FUNCTION_BLOCK "GCS7_E_Maintanance1"	// FB 30
TITLE = Maintenance_1
//  
//COPYRIGHT:    (C) 1997  BUHLER AG, CH-9240 UZWIL, SWITZERLAND
//
//PRODUCT:      GCS7
//
//TITLE:        Element Control Maintenance 1
//
//-------------------------------------------------------------------------
//
//IDENT:        AUTHOR:             DEPT:                       DATE:
//
//FB30.2.2      Ph. Engler          GP92                        31-Jul-2009
//              Flags GCS7_Gr_InMaintWarning and GCS7_Gr_InMaintFault
//FB30.2.1      A. Egli             CT3                         18-Aug-2003
//              FDefineValue 
//FB30.2.0      A. Egli             CT3                         17-Jun-2002
//              New Release with one block 
//FB30.1.1      A.Egli              CT3                         04-Mar-2002
//              Reset CmdFaultReset
//FB30.1.0      A.Egli              CT3                         20-Mar-2000
//              1st Release in S7
//
//-------------------------------------------------------------------------
//
//PURPOSE:      MANUAL : see [MAIN1xxMAN]
//
//RESTRICTIONS: S7
//              ACCU2: Pointer to dynamic datas of the element
//              ACCU1: Pointer to parameter datas of the element
//
//-------------------------------------------------------------------------
//=======================================================
//Log Message: 
//------------------------------------------------------
//1   Counter cleared
//9   fault cancelled
//11  fault 
//12  warning 
//
//=======================================================
//StCode:  State               
//------------------------------------------------------
// 32   StFault        
//  2   StWarning      
//  3   StNormal       
//
//
AUTHOR : EA
FAMILY : GCS7LL
NAME : Maintena
VERSION : 2.2
VAR
  StCode : INT ;	//Element state code
  spare0200 : BOOL ;
  spare0201 : BOOL ;
  spare0202 : BOOL ;
  spare0203 : BOOL ;
  spare0204 : BOOL ;
  InpFault : BOOL ;	//Input to count OutFaultCnt
  InpCount : BOOL ;	//Input to count OutValue
  spare0207 : BOOL ;
  CmdClearValue : BOOL ;	//Clear values
  spare0301 : BOOL ;
  spare0302 : BOOL ;
  CmdFaultReset : BOOL ;	//Command fault reset
  spare0304 : BOOL ;
  spare0305 : BOOL ;
  spare0306 : BOOL ;
  spare0307 : BOOL ;
  OutCopyCount : BOOL ;	//Copy of InpCount
  OutCopyFault : BOOL ;	//Copy of InpFault
  spare0402 : BOOL ;
  spare0403 : BOOL ;
  spare0404 : BOOL ;
  spare0405 : BOOL ;
  spare0406 : BOOL ;
  spare0407 : BOOL ;
  spare0500 : BOOL ;
  spare0501 : BOOL ;
  StNormal : BOOL ;	//OutValue < InWarningValue
  StWarning : BOOL ;	//OutValue >=InWarningValue
  StFault : BOOL ;	//OutValue >=InFaultValue
  spare0505 : BOOL ;
  spare0506 : BOOL ;
  spare0507 : BOOL ;
  InFaultLimit : DINT ;	//Limit for fault           [0.1h] or [number]
  InWarningLimit : DINT ;	//Limit for warning         [0.1h] or [number]
  OutValue : DINT ;	//Actual maintenance value  [0.1h] or [number]
  OutFaultCnt : INT ;	//Number of fault of monitored object [number]
  OutCountSec : INT ;	//Help value to count second
  OutAlarmNrLog : INT ;	//Last textnumber send to log
  Par : STRUCT
   ParObjectNo : INT ;	//Is used for communication with PC, e.g. for message
   ParMsgType : INT ;	//Is used for message (translation of state)
   ParHornCode : INT ;	//Is used by horn module
   ParLogOff : BOOL ;	//Report is off
   ParSpare0401 : BOOL ;
   ParEdgeCnt : BOOL ;	//Type is flag counter
  END_STRUCT ;
END_VAR
VAR_TEMP
  tmpLOGvalue : WORD ;	//LOG value
  tmpLenDyn : DINT ;
  tmpReport : BOOL ;	//Global LOG all
  tmpLocal : BOOL ;
  tmpWarning : BOOL ;
  tmpFault : BOOL ;
END_VAR
BEGIN
NETWORK
TITLE =  Start Global
      L     30;
      T     #tmpLenDyn;	//--> Len dynamic data in byte
NETWORK
TITLE = PC Control
//=== Test Object number =====================
      L     "SYS_DirectCtrlDB".PC.ObjectNo;	//PCControl.ObjectNo
      L     #Par.ParObjectNo;	//Input ObjectNo
      <>I;
      JC    Ctrl;
//=== Test OType      ========================
      L     1830;	//Input object type
      L     "SYS_DirectCtrlDB".PC.ObjectType;	//PCControl.ObjectType
      <>I;
      JC    Ctrl;
//=== Test Handshake =========================
      A     "SYS_DirectCtrlDB".PC.Hsk.FExamine;	// Handshake.FExamine
      JC    pExa;
      A     "SYS_DirectCtrlDB".PC.Hsk.FDefineCmd;	// Handshake.FDefineCmd
      O     "SYS_DirectCtrlDB".PC.Hsk.FDefineValue;	// PC.Hsk.FDefineValue     //[2.1]
      JC    pCmd;
      A     "SYS_DirectCtrlDB".PC.Hsk.FDefinePara;	// Handshake.FDefinePara
      JC    pPar;
pIni: L     2;	// FcInit
      UC    "SYS_DirectCtrl";
      JU    Ctrl;
// Write parameter
pPar: NOP   0;
// Write new commands from PC to Interface of group 
pCmd: A     "SYS_DirectCtrlDB".PC.Cmd1[8];	//Cmd1[8] =CmdClearValue
      S     #CmdClearValue;
      A     "SYS_DirectCtrlDB".PC.Cmd1[11];	//Cmd1[11] =CmdFaultReset
      S     #CmdFaultReset;
//Define Value
      AN    "SYS_DirectCtrlDB".PC.Hsk.FDefineValue;	// PC.Hsk.FDefineValue
      JC    pIni;
      LAR1  P#DBX 58.0;	//PCControl.Value[1]
      L     DBD [AR1,P#6.0];	//PCControl.Value[x+3]
      T     #InFaultLimit;
      L     DBD [AR1,P#10.0];	//PCControl.Value[x+5]
      T     #InWarningLimit;
      JU    pIni;
pExa: TAR2;	// Address Dynamic datas
      T     "SYS_DirectCtrlDB".GC.InDynAddr;	// -->PCControl.GC.InDynAddr
      L     #tmpLenDyn;	// Length Dynamic datas
      T     "SYS_DirectCtrlDB".GC.InDynLen;	// -->PCControl.GC.InDynLen
      L     0;
      T     "SYS_DirectCtrlDB".GC.InParaAddr;	// -->PCControl.GC.InParaAddr
      T     "SYS_DirectCtrlDB".GC.InParaLen;	// -->PCControl.GC.InParaLen
      L     1;	// Code FcExamine
      UC    "SYS_DirectCtrl";
      L     10;	//Revision
      T     "SYS_DirectCtrlDB".GC.Revision;
Ctrl: NOP   0;
NETWORK
TITLE =  All State Init
//---FaultReset is on---
      A     "GCS7_Gr_OutFaultReset";	//Gr.OutFaultReset
      S     #CmdFaultReset;
//===Clear tmp Variable
      AN    #CmdClearValue;
      JC    glJ1;
      L     0;
      T     #OutValue;
      T     #OutFaultCnt;
      T     #OutCountSec;
      O     #Par.ParLogOff;	//---Set LOG Message
      JC    glJ1;
      L     B#(3, 7);	// Message ('Value Cleared' )
      T     #tmpLOGvalue;
      L     W#16#FF;
      AW;
      T     #OutAlarmNrLog;
      CALL  "GCS7_LogConvert" (
           ObjectNo                 := #Par.ParObjectNo,
           MsgType                  := #Par.ParMsgType,
           ClassMsgTxt              := #tmpLOGvalue,
           OType                    := 1030);	// LOG Message Converter / Entry / Contains Class and TextNo
//===Global Group Orders===
//==Count Edges
glJ1: AN    #Par.ParEdgeCnt;
      JC    glJ2;
      A     #InpCount;
      FP    #OutCopyCount;
      JC    glIc;
      JU    glJ4;
//==Running time
glJ2: AN    "GCS7_Gr_OutTick1s";	//Gr.OutTick1s
      ON    #InpCount;
      JC    glJ4;
      L     #OutCountSec;
      +     1;
      T     #OutCountSec;
      L     360;
      <I;
      JC    glJ4;
glIc: L     #OutValue;
      +     L#1;
      T     #OutValue;
      L     0;
      T     #OutCountSec;
//==Count faults
glJ4: NOP   0;
      A     #InpFault;
      FP    #OutCopyFault;
      JCN   glJ5;
      L     #OutFaultCnt;
      +     1;
      T     #OutFaultCnt;
//===Help flags
glJ5: NOP   0;
      L     #OutValue;
      L     #InWarningLimit;
      >=D;
      A(;
      L     0;
      <>D;
      );
      =     #tmpWarning;
      L     #OutValue;
      L     #InFaultLimit;
      >=D;
      A(;
      L     0;
      <>D;
      );
      =     #tmpFault;
NETWORK
TITLE = States
//===State machine===
      A     #StNormal;
      JC    S2;
      A     #StWarning;
      JC    S3;
      A     #StFault;
      JC    S4;
      S     #StNormal;	// Init
      JU    S2;
NETWORK
TITLE = StNormal
// Any transition to StNormal
      S     #StNormal;
      JU    LOG;
//=== Logic ====
//Transition to StFault
S2:   A     #tmpFault;
      R     #StNormal;
      JC    xxS4;
//Transition to StWarning
      A     #tmpWarning;
      R     #StNormal;
      JC    xxS3;
      JU    OUT;
NETWORK
TITLE = StWarning
// Any transition to StWarning
xxS3: S     #StWarning;
      L     B#(1, 12);	// Message ('Warning')
      JU    LOG;
//=== Logic ====
// Transition to StFault
S3:   A     #tmpFault;
      R     #StWarning;
      JC    xxS4;
//  Retry message
      A     #CmdFaultReset;
      O     "GCS7_Gr_OutFaultReset";	// OutFaultReset
      A     #tmpWarning;
      JC    xxS3;
// Transition to StNormal
      A     #tmpWarning;
      JC    OUT;
      R     #StWarning;
      S     #StNormal;
      L     B#(3, 9);	// Message ('fault cancelled' )
      JU    LOG;
NETWORK
TITLE = StFault
// Any transiton to Fault  
xxS4: S     "GCS7_Gr_InFaultFlag";	// Gr.InFaultFlag
      S     #StFault;
      CALL  "SYS_Horn_Code" (
           FcCode                   := 1,
           ParObjectType            := 1030,
           ParObjectNo              := #Par.ParObjectNo,
           ParHornCode              := #Par.ParHornCode);
      L     B#(1, 11);	// Message ('fault')
      JU    LOG;
//=== Logic ====
// retry of fault message
S4:   A     #CmdFaultReset;
      O     "GCS7_Gr_OutFaultReset";	//Gr.OutFaultReset
      A     #tmpFault;
      L     B#(1, 11);	// Message ('fault')
      JC    LOG;
      A     #tmpFault;
      JC    OUT;
      R     #StFault;
      S     #StNormal;
      L     B#(3, 9);	// Message ('fault cancelled' )
      JU    LOG;
NETWORK
TITLE = LOG
LOG:  A     #Par.ParLogOff;	//---Set LOG Message
      JC    OUT;
      T     #tmpLOGvalue;
      L     W#16#FF;
      AW;
      T     #OutAlarmNrLog;
      CALL  "GCS7_LogConvert" (
           ObjectNo                 := #Par.ParObjectNo,
           MsgType                  := #Par.ParMsgType,
           ClassMsgTxt              := #tmpLOGvalue,
           OType                    := 1030);	// LOG Message Converter / Entry / Contains Class and TextNo
NETWORK
TITLE = Global End
OUT:  SET;
      R     #CmdClearValue;
      R     #CmdFaultReset;	//[1.1]
// 
      A     #StWarning;	//[2.2]
      S     "GCS7_Gr_InMaintWarning";	//[2.2]
      A     #StFault;	//[2.2]
      S     "GCS7_Gr_InMaintFault";	//[2.2]
NETWORK
TITLE = State Code
      L     2;	// Code: Warning
      A     #StWarning;
      JC    STC;
      L     3;	// Code: Normal
      A     #StNormal;
      JC    STC;
      L     32;	// Code: fault
STC:  L     #StCode;	// Old state code
      TAK;
      T     #StCode;	// Save state code
      <>I;
      L     3;	// Load code for CBit methode
      CC    "SYS_CBitCtrl";
END_FUNCTION_BLOCK

FUNCTION_BLOCK "GCS7_E_Maintanance2"	// FB 31
TITLE = Maintenance_2
//  
//COPYRIGHT:    (C) 1997  BUHLER AG, CH-9240 UZWIL, SWITZERLAND
//
//PRODUCT:      GCS7
//
//TITLE:        Element Control Maintenance 2
//
//-------------------------------------------------------------------------
//
//IDENT:        AUTHOR:             DEPT:                       DATE:
//
//FB31.2.2      Ph. Engler          GP92                        31-Jul-2009
//              Flags GCS7_Gr_InMaintWarning and GCS7_Gr_InMaintFault
//FB31.2.1      A. Egli             CT3                         18-Aug-2003
//              FDefineValue
//FB31.2.0      A. Egli             CT3                         17-Jun-2002
//              New Release with one block 
//FB31.1.1      A.Egli              CT3                         04-Mar-2002
//              Reset CmdFaultReset
//FB31.1.0      A.Egli              CT3                         20-Mar-2000
//              1st Release in S7
//
//-------------------------------------------------------------------------
//
//PURPOSE:      MANUAL : see [MAIN2xxMAN]
//                
//
//RESTRICTIONS: S7
//              ACCU2: Pointer to dynamic datas of the element
//              ACCU1: Pointer to parameter datas of the element
//
//-------------------------------------------------------------------------
//=======================================================
//Log Message: 
//------------------------------------------------------
// 1   Counter cleared
// 9   fault cancelled
//11   fault 
//12   warning 
//
//
//=======================================================
//StCode:  State               
//------------------------------------------------------
// 32   StFault        
//  2   StWarning      
//  3   StNormal       
//
AUTHOR : EA
FAMILY : GCS7LL
NAME : Maintena
VERSION : 2.2
VAR
  StCode : INT ;	//Element state code
  spare0200 : BOOL ;
  spare0201 : BOOL ;
  spare0202 : BOOL ;
  spare0203 : BOOL ;
  spare0204 : BOOL ;
  InpFault : BOOL ;	//Input to count fault values
  InpRun : BOOL ;	//Input to count running times
  spare0207 : BOOL ;
  CmdClearValue : BOOL ;	//Clear maintenance values
  CmdClearTotalValue : BOOL ;	//Clear maintenance values and total hours
  spare0302 : BOOL ;
  CmdFaultReset : BOOL ;	//Command fault reset
  spare0304 : BOOL ;
  spare0305 : BOOL ;
  spare0306 : BOOL ;
  spare0307 : BOOL ;
  OutCopyFault : BOOL ;	//Copy of InpFault
  spare0401 : BOOL ;
  spare0402 : BOOL ;
  spare0403 : BOOL ;
  spare0404 : BOOL ;
  spare0405 : BOOL ;
  spare0406 : BOOL ;
  spare0407 : BOOL ;
  spare0500 : BOOL ;
  spare0501 : BOOL ;
  StNormal : BOOL ;	//OutValue < InWarningValue
  StWarning : BOOL ;	//OutValue >=InWarningValue
  StFault : BOOL ;	//OutValue >=InFaultValue
  spare0505 : BOOL ;
  spare0506 : BOOL ;
  spare0507 : BOOL ;
  InFaultLimit : DINT ;	//Limit for fault      [0.1 h]
  InWarningLimit : DINT ;	//Limit for warning    [0.1 h]
  OutTotalHours : DINT ;	//Running hours since last maintenance [0.1 h]
  OutMaintenanceHours : DINT ;	//Running hours since last maintenance [0.1 h]
  OutFaultHours : DINT ;	//Fault hours since last maintenance [0.1 h]
  OutFaultCounter : INT ;
  OutResetDate : STRUCT 	//Last maintenance
   Year : INT ;
   Month : BYTE ;
   Day : BYTE ;
   Hour : BYTE ;
   Min : BYTE ;
  END_STRUCT ;
  OutTotalSec : INT ;	//Help value to count seconds
  OutMaintenanceSec : INT ;	//Help value to count seconds
  OutFaultSec : INT ;	//Help value to count seconds
  OutAlarmNrLog : INT ;	//Last textnumber send to log
  Par : STRUCT
   ParObjectNo : INT ;	//Is used for communication with PC, e.g. for message
   ParMsgType : INT ;	//Is used for message (translation of state)
   ParHornCode : INT ;	//Is used by horn module
   ParLogOff : BOOL ;	//Report is off
  END_STRUCT ;
END_VAR
VAR_TEMP
  tmpLOGvalue : WORD ;	//LOG value
  tmpLenDyn : DINT ;
  tmpReport : BOOL ;	//Global LOG all
  tmpLocal : BOOL ;
  tmpWarning : BOOL ;
  tmpFault : BOOL ;
  tmpDateTime : DATE_AND_TIME ;
  tmpRet : INT ;
END_VAR
BEGIN
NETWORK
TITLE =  Start Global
      L     48;
      T     #tmpLenDyn;	//--> Len dynamic data in byte
NETWORK
TITLE = PC Control
//=== Test Object number =====================
      L     "SYS_DirectCtrlDB".PC.ObjectNo;	//PCControl.ObjectNo
      L     #Par.ParObjectNo;	//Input ObjectNo
      <>I;
      JC    Ctrl;
//=== Test OType      ========================
      L     1831;	//Input object type
      L     "SYS_DirectCtrlDB".PC.ObjectType;	//PCControl.ObjectType
      <>I;
      JC    Ctrl;
//=== Test Handshake =========================
      A     "SYS_DirectCtrlDB".PC.Hsk.FExamine;	// Handshake.FExamine
      JC    pExa;
      A     "SYS_DirectCtrlDB".PC.Hsk.FDefineCmd;	// Handshake.FDefineCmd
      O     "SYS_DirectCtrlDB".PC.Hsk.FDefineValue;	// Handshake.FDefineValue  //[2.1]
      JC    pCmd;
      A     "SYS_DirectCtrlDB".PC.Hsk.FDefinePara;	// Handshake.FDefinePara
      JC    pPar;
pIni: L     2;	// FcInit
      UC    "SYS_DirectCtrl";
      JU    Ctrl;
// Write parameter
pPar: NOP   0;
// Write new commands from PC to Interface of group 
pCmd: A     "SYS_DirectCtrlDB".PC.Cmd1[8];	//Cmd1[8] =CmdClearValue
      S     #CmdClearValue;
      A     "SYS_DirectCtrlDB".PC.Cmd1[9];	//Cmd1[8] =CmdClearValue
      S     #CmdClearTotalValue;
      A     "SYS_DirectCtrlDB".PC.Cmd1[11];	//Cmd1[11] =CmdFaultReset
      S     #CmdFaultReset;
//Define Value
      AN    "SYS_DirectCtrlDB".PC.Hsk.FDefineValue;	// PC.Hsk.FDefineValue
      JC    pIni;
      LAR1  P#DBX 58.0;	//PCControl.Value[1]
      L     DBD [AR1,P#6.0];	//PCControl.Value[x+3]
      T     #InFaultLimit;
      L     DBD [AR1,P#10.0];	//PCControl.Value[x+5]
      T     #InWarningLimit;
      JU    pIni;
pExa: TAR2;	// Address Dynamic datas
      T     "SYS_DirectCtrlDB".GC.InDynAddr;	// -->PCControl.GC.InDynAddr
      L     #tmpLenDyn;	// Length Dynamic datas
      T     "SYS_DirectCtrlDB".GC.InDynLen;	// -->PCControl.GC.InDynLen
      L     0;
      T     "SYS_DirectCtrlDB".GC.InParaAddr;	// -->PCControl.GC.InParaAddr
      T     "SYS_DirectCtrlDB".GC.InParaLen;	// -->PCControl.GC.InParaLen
      L     1;	// Code FcExamine
      UC    "SYS_DirectCtrl";
      L     10;	//Revision
      T     "SYS_DirectCtrlDB".GC.Revision;
Ctrl: NOP   0;
NETWORK
TITLE =  All State Init
//---FaultReset is on--
      A     "GCS7_Gr_OutFaultReset";	//Gr.OutFaultReset
      S     #CmdFaultReset;
//===Clear tmp Variable
      AN    #CmdClearTotalValue;
      JC    glR0;
      L     0;
      T     #OutTotalHours;
      T     #OutTotalSec;
      O     #Par.ParLogOff;	//---Set LOG Message
      JC    glR0;
      L     B#(3, 8);	// Message ('Total Value Cleared' )
      T     #tmpLOGvalue;
      L     W#16#FF;
      AW;
      T     #OutAlarmNrLog;
      CALL  "GCS7_LogConvert" (
           ObjectNo                 := #Par.ParObjectNo,
           MsgType                  := #Par.ParMsgType,
           ClassMsgTxt              := #tmpLOGvalue,
           OType                    := 1031);	// LOG Message Converter / Entry / Contains Class and TextNo
//===Clear tmp Variable
glR0: AN    #CmdClearValue;
      JC    glJ1;
      CALL  "SIEMENS_READ_CLK" (
           RET_VAL                  := #tmpRet,
           CDT                      := #tmpDateTime);
      LAR1  P##tmpDateTime;
      L     1900;
      L     LB [AR1,P#0.0];
      BTI;
      +I;
      L     1990;
      >=I;
      TAK;
      JC    glJa;
      +     100;
glJa: T     #OutResetDate.Year;
      L     LB [AR1,P#1.0];
      BTI;
      T     #OutResetDate.Month;
      L     LB [AR1,P#2.0];
      BTI;
      T     #OutResetDate.Day;
      L     LB [AR1,P#3.0];
      BTI;
      T     #OutResetDate.Hour;
      L     LB [AR1,P#4.0];
      BTI;
      T     #OutResetDate.Min;
      L     #OutMaintenanceHours;
      L     0;
      ==D;
      T     #OutMaintenanceHours;
      T     #OutFaultHours;
      T     #OutFaultCounter;
      T     #OutMaintenanceSec;
      T     #OutFaultSec;
      O     #Par.ParLogOff;	//---Set LOG Message
      JC    glJ1;
      L     B#(3, 7);	// Message ('Value Cleared' )
      T     #tmpLOGvalue;
      L     W#16#FF;
      AW;
      T     #OutAlarmNrLog;
      CALL  "GCS7_LogConvert" (
           ObjectNo                 := #Par.ParObjectNo,
           MsgType                  := #Par.ParMsgType,
           ClassMsgTxt              := #tmpLOGvalue,
           OType                    := 1031);	// LOG Message Converter / Entry / Contains Class and TextNo
//===Global Group Orders===
// Count Faults
glJ1: A     #InpFault;
      FP    #OutCopyFault;
      JCN   glJ2;
      L     #OutFaultCounter;
      +     L#1;
      T     #OutFaultCounter;
// Count Fault time
glJ2: AN    "GCS7_Gr_OutTick1s";	//Gr.OutTick1s
      ON    #InpFault;
      JC    glJ3;
      L     #OutFaultSec;
      +     1;
      T     #OutFaultSec;
      L     360;
      <I;
      JC    glJ3;
      L     #OutFaultHours;
      +     L#1;
      T     #OutFaultHours;
      L     0;
      T     #OutFaultSec;
//Maintenance hour
glJ3: AN    "GCS7_Gr_OutTick1s";	//Gr.OutTick1s
      ON    #InpRun;
      JC    glJ4;
      L     #OutMaintenanceSec;
      +     1;
      T     #OutMaintenanceSec;
      L     360;
      <I;
      JC    glJ4;
      L     #OutMaintenanceHours;
      +     L#1;
      T     #OutMaintenanceHours;
      L     0;
      T     #OutMaintenanceSec;
//Total hour
glJ4: AN    "GCS7_Gr_OutTick1s";	//Gr.OutTick1s
      ON    #InpRun;
      JC    glJ5;
      L     #OutTotalSec;
      +     1;
      T     #OutTotalSec;
      L     360;
      <I;
      JC    glJ5;
      L     #OutTotalHours;
      +     L#1;
      T     #OutTotalHours;
      L     0;
      T     #OutTotalSec;
//Help Flags
glJ5: L     #OutMaintenanceHours;
      L     #InWarningLimit;
      >=D;
      A(;
      L     0;
      <>D;
      );
      =     #tmpWarning;
      L     #OutMaintenanceHours;
      L     #InFaultLimit;
      >=D;
      A(;
      L     0;
      <>D;
      );
      =     #tmpFault;
NETWORK
TITLE = States
//===State machine===
      A     #StNormal;
      JC    S2;
      A     #StWarning;
      JC    S3;
      A     #StFault;
      JC    S4;
      S     #StNormal;	// Init
      JU    S2;
NETWORK
TITLE = StNormal
// Any transition to StNormal
      S     #StNormal;
      JU    LOG;
//=== Logic ====
//Transition to StFault
S2:   A     #tmpFault;
      R     #StNormal;
      JC    xxS4;
//Transition to StWarning
      A     #tmpWarning;
      R     #StNormal;
      JC    xxS3;
      JU    OUT;
NETWORK
TITLE = StWarning
// Any transition to StWarning
xxS3: S     #StWarning;
      L     B#(1, 12);	// Message ('Warning')
      JU    LOG;
//=== Logic ====
// Transition to StFault
S3:   A     #tmpFault;
      R     #StWarning;
      JC    xxS4;
//  Retry message
      A     #CmdFaultReset;
      O     "GCS7_Gr_OutFaultReset";	// OutFaultReset
      A     #tmpWarning;
      JC    xxS3;
// Transition to StNormal
      A     #tmpWarning;
      JC    OUT;
      R     #StWarning;
      S     #StNormal;
      L     B#(3, 9);	// Message ('fault cancelled' )
      JU    LOG;
NETWORK
TITLE = StFault
// Any transiton to Fault  
xxS4: S     "GCS7_Gr_InFaultFlag";	// Gr.InFaultFlag
      S     #StFault;
      CALL  "SYS_Horn_Code" (
           FcCode                   := 1,
           ParObjectType            := 1031,
           ParObjectNo              := #Par.ParObjectNo,
           ParHornCode              := #Par.ParHornCode);
      L     B#(1, 11);	// Message ('fault')
      JU    LOG;
//=== Logic ====
// retry of fault message
S4:   A     #CmdFaultReset;
      O     "GCS7_Gr_OutFaultReset";	//Gr.OutFaultReset
      A     #tmpFault;
      L     B#(1, 11);	// Message ('fault')
      JC    LOG;
      A     #tmpFault;
      JC    OUT;
      R     #StFault;
      S     #StNormal;
      L     B#(3, 9);	// Message ('fault cancelled' )
      JU    LOG;
NETWORK
TITLE = LOG
LOG:  A     #Par.ParLogOff;	//---Set LOG Message
      JC    OUT;
      T     #tmpLOGvalue;
      L     W#16#FF;
      AW;
      T     #OutAlarmNrLog;
      CALL  "GCS7_LogConvert" (
           ObjectNo                 := #Par.ParObjectNo,
           MsgType                  := #Par.ParMsgType,
           ClassMsgTxt              := #tmpLOGvalue,
           OType                    := 1031);	// LOG Message Converter / Entry / Contains Class and TextNo
NETWORK
TITLE = Global End
OUT:  SET;
      R     #CmdClearValue;
      R     #CmdClearTotalValue;
      R     #CmdFaultReset;	//[1.1]
// 
      A     #StWarning;	//[2.2]
      S     "GCS7_Gr_InMaintWarning";	//[2.2]
      A     #StFault;	//[2.2]
      S     "GCS7_Gr_InMaintFault";	//[2.2]
NETWORK
TITLE = State Code
      L     2;	// Code: Warning
      A     #StWarning;
      JC    STC;
      L     3;	// Code: Normal
      A     #StNormal;
      JC    STC;
      L     32;	// Code: fault
STC:  L     #StCode;	// Old state code
      TAK;
      T     #StCode;	// Save state code
      <>I;
      L     3;	// Load code for CBit methode
      CC    "SYS_CBitCtrl";
END_FUNCTION_BLOCK

FUNCTION_BLOCK "GCS7_E_MZAF"	// FB 32
TITLE = Flowbalancer MZAF
//  
//COPYRIGHT:    (C) 1997  BUHLER AG, CH-9240 UZWIL, SWITZERLAND
//
//PRODUCT:      GCS7
//
//TITLE:        Element Control MZAF
//
//-------------------------------------------------------------------------
//
//IDENT:        AUTHOR:             DEPT:                       DATE:
//
//FB32.3.0      A. Egli             CT3                         17-Jun-2002
//              New Release with one block 
//FB32.2.1      A. Egli             CT3                         11-Oct-1999
//              M12.2 "Gr.OutCmdNext removed
//FB32.2A       A. Egli             CT3                         04-Mai-1998
//              StFault = StCode 32
//FB32.1A       A.Egli              AEE61                       31-Jul-1997
//              1st Release in S7
//
//-------------------------------------------------------------------------
//
//PURPOSE:      MANUAL : see [MZAxxMAN]
//
//RESTRICTIONS: S7
//              ACCU2: Pointer to dynamic datas of the element
//              ACCU1: Pointer to parameter datas of the element
//
//-------------------------------------------------------------------------
//
//=======================================================
//Log Message: 
//------------------------------------------------------
// 0   stopped
// 1   started
// 9   fault cancelled
//10  fault adjust
//
//=======================================================
//StCode:  State               
//------------------------------------------------------
//32   StFault                 
// 1   StStopped                    Stopped
//41   Stopped.HWStop               StStopped + InHWStop 
//51   Stopped.DPFault              StStopped + DPFault
// 2   StAdjusting             
// 3   StStarted               
//
//
//
AUTHOR : EA
FAMILY : GCS7LL
NAME : MZAF
VERSION : 3.0
VAR
  StCode : INT ;	//Element state code
  InEnable : BOOL ;	//Enable to run
  spare0201 : BOOL ;
  spare0202 : BOOL ;
  spare0203 : BOOL ;
  spare0204 : BOOL ;
  CmdNewJob : BOOL ;	//Pulse to erase OutJobWeight
  InFlapOpen : BOOL ;	//Flap is open, command to count up OutJobWeight
  InpAdjusted : BOOL ;	//Digital input element is adjusted
  CmdOff : BOOL ;	//Pulse to start in manual mode
  CmdOn : BOOL ;	//Pulse to stop in manual mode
  CmdNext : BOOL ;	//Start next element (Automatic mode)
  CmdFaultReset : BOOL ;	//Command to reset fault
  InLocal : BOOL ;	//1= Local mode
  InManual : BOOL ;	//1= Manual/ 0= Automatic
  InReport : BOOL ;	//Report of all state transitions
  spare0307 : BOOL ;
  InHWStop : BOOL ;	//ALL : HW stop is detected, no fault
  InDPFault : BOOL ;	//ALL : DP-Fault is detected, no fault
  spare0402 : BOOL ;
  spare0403 : BOOL ;
  spare0404 : BOOL ;
  spare0405 : BOOL ;
  spare0406 : BOOL ;
  OutpAirValve : BOOL ;	//Digital output air valve
  StStopped : BOOL ;	//Element is stopped
  StAdjusting : BOOL ;	//Element is adjusting
  StStarted : BOOL ;	//Element is adjusted
  spare0503 : BOOL ;
  StFault : BOOL ;	//Element has a fault
  InOutFlowratePpm : INT ;	//Flowrate target value in [0.1 %]
  InOutFlowrate : DINT ;	//Flowrate target value in [kg/h]
  OutJobWeight : DINT ;	//Total feeded weight [kg]
  OutpFlowrate : INT ;	//Analog value to set flowrate [digits]
  OutAlarmNrLog : INT ;	//Last textnumber send to log
  Par : STRUCT
   ParObjectNo : INT ;	//Is used for communication with PC, e.g. for message
   ParMsgType : INT ;	//Is used for message (translation of state)
   ParHornCode : INT ;	//Is used by horn module
   ParLogOff : BOOL ;	//Report is off
   ParManual : BOOL ;	//Manual mode without interlocking
   ParFlowratePc : BOOL ;	//Target value for flowrate in Pc
   ParSpare0403 : BOOL ;
   ParWago : BOOL ;	//Wago analog module format
   ParMonTime : INT ;	//After this time the element must be adjusted [0.1 s]
   ParFlowrate100Pc : DINT  := L#10000;	//Flow rate by 100 % of analog output [kg/h]
   OutMonTime : INT  := 100;	//Actual monitoring time [0.1 s]
   OutWtCorrection : REAL ;	//Correction weight for calcuation of OutWtTotal [kg]
  END_STRUCT ;
END_VAR
VAR_TEMP
  tmpLOGvalue : WORD ;	//LOG value
  tmpLenDyn : DINT ;
  tmpReport : BOOL ;	//Global LOG all
  tmpEnable : BOOL ;
  tmpEndTime : BOOL ;
  tmpLocal : BOOL ;
  tmpMaxDigits : REAL ;	//ParWago=0: 27'648 / ParWago=1: 32'767
  tmpLocalFault : BOOL ;
END_VAR
BEGIN
NETWORK
TITLE =  Start Global
      L     38;
      T     #tmpLenDyn;	//--> Len dynamic data in byte
NETWORK
TITLE = PC Control
//=== Test Object number =====================
      L     "SYS_DirectCtrlDB".PC.ObjectNo;	//PCControl.ObjectNo
      L     #Par.ParObjectNo;	//Input ObjectNo
      <>I;
      JC    Ctrl;
//=== Test OType      ========================
      L     1032;	//Input object type
      L     "SYS_DirectCtrlDB".PC.ObjectType;	//PCControl.ObjectType
      <>I;
      JC    Ctrl;
//=== Test Handshake =========================
      A     "SYS_DirectCtrlDB".PC.Hsk.FExamine;	// Handshake.FExamine
      JC    pExa;
      A     "SYS_DirectCtrlDB".PC.Hsk.FDefineCmd;	// Handshake.FDefineCmd
      JC    pCmd;
      A     "SYS_DirectCtrlDB".PC.Hsk.FDefinePara;	// Handshake.FDefinePara
      JC    pPar;
pIni: L     2;	// FcInit
      UC    "SYS_DirectCtrl";
      JU    Ctrl;
// Write parameter 
pPar: LAR1  P#DBX 58.0;	//PCControl.Value[1]
      L     #tmpLenDyn;
      SLD   3;
      +AR1;
      L     DBW [AR1,P#8.0];	//PCControl.Value
      T     #Par.ParMonTime;
// Write new commands from PC to Interface of group 
pCmd: A     "SYS_DirectCtrlDB".PC.Cmd1[8];	//Cmd1[8] =CmdOff
      S     #CmdOff;
      A     "SYS_DirectCtrlDB".PC.Cmd1[9];	//Cmd1[9] =CmdOn
      S     #CmdOn;
      A     "SYS_DirectCtrlDB".PC.Cmd1[10];	//Cmd1[10] =CmdNext
      S     #CmdNext;
      A     "SYS_DirectCtrlDB".PC.Cmd1[11];	//Cmd1[11] =CmdFaultReset
      S     #CmdFaultReset;
      A     "SYS_DirectCtrlDB".PC.Cmd1[13];	//Cmd1[13] =CmdManualOn
      S     #InManual;
      A     "SYS_DirectCtrlDB".PC.Cmd2[13];	//Cmd2[13] =CmdManualOff
      R     #InManual;
      A     "SYS_DirectCtrlDB".PC.Cmd1[14];	//Cmd1[14]=CmdReportOn
      S     #InReport;
      A     "SYS_DirectCtrlDB".PC.Cmd2[14];	//Cmd2[14]=CmdReportOff
      R     #InReport;
//Define Value
      AN    "SYS_DirectCtrlDB".PC.Hsk.FDefineValue;	// PC.Hsk.FDefineValue
      ON    #InManual;
      JC    pIni;
      LAR1  P#DBX 58.0;
      L     DBW [AR1,P#6.0];
      T     #InOutFlowratePpm;
      L     DBD [AR1,P#8.0];
      T     #InOutFlowrate;
      JU    pIni;
pExa: TAR2;	// Address Dynamic datas
      T     "SYS_DirectCtrlDB".GC.InDynAddr;	// -->PCControl.GC.InDynAddr
      L     #tmpLenDyn;	// Length Dynamic datas
      T     "SYS_DirectCtrlDB".GC.InDynLen;	// -->PCControl.GC.InDynLen
      L     0;
      T     "SYS_DirectCtrlDB".GC.InParaAddr;	// -->PCControl.GC.InParaAddr
      T     "SYS_DirectCtrlDB".GC.InParaLen;	// -->PCControl.GC.InParaLen
      L     1;	// Code FcExamine
      UC    "SYS_DirectCtrl";
      L     10;	//Revision
      T     "SYS_DirectCtrlDB".GC.Revision;
NETWORK
TITLE =  All State Init
//===Clear tmp Variable
//===Global Group Orders===
Ctrl: A     "GCS7_Gr_OutManualOn";	//Gr.OutManualOn
      S     #InManual;
      A     "GCS7_Gr_OutManualOff";	//Gr.OutManualOff
      R     #InManual;
      A     #InManual;
      S     "GCS7_Gr_InManual";	//Gr.InManualMode
//---Local---
      A     #InLocal;
      AN    #InManual;
      =     #tmpLocalFault;
      A     #tmpLocalFault;
      O     #InHWStop;
      O     #InDPFault;
      =     #tmpLocal;
//---Report is on---
      A     "GCS7_Gr_OutReportAll";	//Gr.OutReportAll
      O     #InReport;
      =     #tmpReport;
//---tmpEnable---
      A     #InEnable;
      AN    #InLocal;
      AN    #InManual;
      O(;
      A     #InEnable;
      O     #Par.ParManual;
      A     #InManual;
      );
      AN    #CmdOff;
      =     #tmpEnable;
//---tmpMaxDigits
      L     2.764800e+04;	//Siemens fullrange MaxDigits
      AN    #Par.ParWago;
      JC    Ctr2;
      L     3.276700e+04;	//Wago fullrange MaxDigits
Ctr2: T     #tmpMaxDigits;
NETWORK
TITLE = States
//===State machine===
      A     #StStopped;
      JC    S0;
      A     #StAdjusting;
      JC    S1;
      A     #StStarted;
      JC    S2;
      A     #StFault;
      JC    S4;
      S     #StStopped;	// Init    
      JU    S0;
NETWORK
TITLE = StStopped
// Any transition to StStopped
xxS0: S     #StStopped;
      AN    #InReport;
      JC    OUT;
      L     B#(4, 0);	// Message ('stopped' )
      JU    LOG;
//=== Logic ====
//Transition to StStarted 
S0:   A     #CmdNext;
      AN    #InManual;
      A     #tmpEnable;
      O;
      A     #CmdOn;
      A     #InManual;
      A     #tmpEnable;
      R     #StStopped;
      JC    xxS2;
      JU    OUT;
NETWORK
TITLE = StAdjusting
// Any transition to StAdjusting
xxS1: S     #StAdjusting;
      L     0;
      T     #Par.OutMonTime;
      JU    OUT;
//=== Logic ====
S1:   AN    "GCS7_Gr_OutTick1s";	//Gr.OutTick1s
      O     #tmpLocal;
      L     #Par.OutMonTime;
      JC    S1J3;
      +     10;
      T     #Par.OutMonTime;
S1J3: L     #Par.ParMonTime;
      >=I;
      =     #tmpEndTime;
// Transition to StStopped
      AN    #tmpEnable;
      R     #StAdjusting;
      JC    xxS0;
// Transition to StStarted
      A     #InpAdjusted;
      R     #StAdjusting;
      JC    xxS2;
// Transition to StFault
      A     #tmpEndTime;
      AN    #tmpLocal;
      R     #StAdjusting;
      JC    xxS4;
      JU    OUT;
NETWORK
TITLE = StStarted
// Any transition to StStarted
xxS2: S     #StStarted;
      S     #StStarted;
      AN    #tmpReport;
      JC    OUT;
      L     B#(4, 1);	// Message ('started')
      JU    LOG;
//=== Logic ====
//Transition to StStopped
S2:   AN    #tmpEnable;
      R     #StStarted;
      JC    xxS0;
//Transition to StAdjusting
      AN    #InpAdjusted;
      R     #StStarted;
      JC    xxS1;
      JU    OUT;
NETWORK
TITLE = StFault
// Any transiton to Fault  
xxS4: S     "GCS7_Gr_InFaultFlag";	// Gr.InFaultFlag
      S     #StFault;
      CALL  "SYS_Horn_Code" (
           FcCode                   := 1,
           ParObjectType            := 1032,
           ParObjectNo              := #Par.ParObjectNo,
           ParHornCode              := #Par.ParHornCode);
      L     B#(1, 10);	// Message ('fault adjust')
      JU    LOG;
//=== Logic ====
S4:   AN    #CmdFaultReset;
      AN    "GCS7_Gr_OutFaultReset";	//  Gr.OutFaultReset
      AN    #tmpLocalFault;
      JC    OUT;
// retry of fault message
      AN    #InpAdjusted;
      AN    #tmpLocal;
      JC    xxS4;
      R     #StFault;
      S     #StStopped;
      L     B#(3, 9);	// Message ('fault cancelled' )
      JU    LOG;
NETWORK
TITLE = LOG
LOG:  A     #Par.ParLogOff;	//---Set LOG Message
      JC    OUT;
      T     #tmpLOGvalue;
      L     W#16#FF;
      AW;
      T     #OutAlarmNrLog;
      CALL  "GCS7_LogConvert" (
           ObjectNo                 := #Par.ParObjectNo,
           MsgType                  := #Par.ParMsgType,
           ClassMsgTxt              := #tmpLOGvalue,
           OType                    := 1032);	// LOG Message Converter / Entry / Contains Class and TextNo
NETWORK
TITLE = Calculate Flow rate
OUT:  A     #Par.ParFlowratePc;
      JC    frPc;
      L     #InOutFlowrate;
      DTR;
      L     #Par.ParFlowrate100Pc;
      DTR;
      /R;
      L     1.000000e+03;
      *R;
      RND;
      T     #InOutFlowratePpm;
      JU    avJ0;
frPc: L     #InOutFlowratePpm;
      DTR;
      L     1.000000e+03;
      /R;
      L     #Par.ParFlowrate100Pc;
      DTR;
      *R;
      RND;
      T     #InOutFlowrate;
NETWORK
TITLE = Calculate Analog value
avJ0: L     0;
      A     #StFault;
      JC    avJ1;
      L     #InOutFlowrate;	// kg/h    
      DTR;	// Integer to real
      L     #Par.ParFlowrate100Pc;
      DTR;	// Integer to real
      <=R;
      JC    avJ2;
      L     1.000000e+00;	// 100%          
      JU    avJ3;
avJ2: /R;
avJ3: L     #tmpMaxDigits;	// Units maximum
      *R;
      RND;	// Real to Integer
avJ1: T     #OutpFlowrate;
NETWORK
TITLE = Calculate OutWtTotal
      AN    #CmdNewJob;
      JC    wtJ1;
      L     0;
      T     #OutJobWeight;
      L     0.000000e+00;
      T     #Par.OutWtCorrection;
      JU    clJ1;
wtJ1: ON    #InFlapOpen;
      ON    "GCS7_Gr_OutTick1s";	//Gr.OutTick1s
      JC    clJ1;
      L     #InOutFlowrate;
      DTR;	// Integer to Real
      L     3.600000e+03;	// [3600s]  
      /R;
      L     #Par.OutWtCorrection;
      +R;
      T     #Par.OutWtCorrection;
      RND-;
      L     #OutJobWeight;
      +D;
      T     #OutJobWeight;
      L     #Par.OutWtCorrection;
      L     #Par.OutWtCorrection;
      RND-;
      DTR;	// Integer to Real
      -R;
      T     #Par.OutWtCorrection;	//New rest 
//---Clear all commands
NETWORK
TITLE = Global End
clJ1: SET;
      R     #CmdOn;
      R     #CmdOff;
      R     #CmdNewJob;
      R     #CmdFaultReset;
      R     #CmdNext;
//---Digital output
      A     #StStarted;
      O     #StAdjusting;
      =     #OutpAirValve;
//--Output for group 
      AN    #InLocal;
      O     #InManual;
      A     #InDPFault;
      S     "GCS7_Gr_InDPFault";
      AN    #InLocal;
      O     #InManual;
      A     #InHWStop;
      S     "GCS7_Gr_InHWStop";
NETWORK
TITLE = State Code
//--Stopped, Substate ---
      AN    #StStopped;
      JC    STC2;
      L     41;	//Code: StStopped.HWStop
      A     #InHWStop;
      JC    STC;
      L     51;	//Code: StStopped.DPFault
      A     #InDPFault;
      JC    STC;
      L     1;	// Code: stopped
      JC    STC;
//--------------------
STC2: L     2;	// Code: adjusting
      A     #StAdjusting;
      JC    STC;
      L     3;	// Code: started
      A     #StStarted;
      JC    STC;
      L     32;	// Code: fault
STC:  L     #StCode;	// Old state code    
      TAK;
      T     #StCode;	// Save state code    
      <>I;
      L     3;	// Load code for CBit methode
      CC    "SYS_CBitCtrl";
END_FUNCTION_BLOCK

FUNCTION_BLOCK "GCS7_E_MYAH"	// FB 33
TITLE = MYAH
//  
//COPYRIGHT:    (C) 2004 BY  BUHLER AG, CH-9240 UZWIL  SWITZERLAND
//
//PRODUCT:      GCS7
//
//TITLE:        Element MYAH Yield PC (Profibus)
//              (GCPROVB Revision 10)
//
//-------------------------------------------------------------------------
//
//IDENT:        AUTHOR:             DEPT:                      DATE:
//FB33.1.0      A. Egli             CT3                        08-Jan-2006
//              1st Release in S7
//
//-------------------------------------------------------------------------
//
//PURPOSE:      MANUAL : see [MYAHENMAN]
//
//RESTRICTIONS: S7
//
//              (*2) : Not used for MZDE
//
//=======================================================
//Log Message: 
//------------------------------------------------------
//0     = Fault Cannceled
//1..79 = AlarmLC : Alarmnumber see manual of MEAF
//90    = Fault Remote Control
//91    = StStopped
//92    = StDosing
//93    = StEmptied
//94    = Timeout starting
//95    = Wrong value
//96    = Communication fault
//97    = 
//98    = 
//99    = Collected alarm
//
//=======================================================
//StCode:  State               
//------------------------------------------------------
//32    StFault                 
// 1    StStopped                   Stopped
//41    Stopped.HWStop              StStopped + InHWStop 
//51    Stopped.DPFault             StStopped + DPFault
// 2    StStarting              
// 3    StStarted               
// 7    StStopping              
//
//
AUTHOR : EA
FAMILY : GCS7LL
NAME : MYAH
VERSION : 1.0
VAR
  StCode : INT ;	//Element state code
  InEnable : BOOL ;	//Enable to run the element (manual and automatic mode)
  spare0201 : BOOL ;
  spare0202 : BOOL ;
  spare0203 : BOOL ;
  spare0204 : BOOL ;
  spare0205 : BOOL ;
  spare0206 : BOOL ;
  spare0207 : BOOL ;
  CmdOff : BOOL ;	//Pulse to stop the element (manual mode)
  CmdOn : BOOL ;	//Pulse to start the element (manual mode)
  CmdNext : BOOL ;	//Pulse to start the element in automatic mode
  CmdFaultReset : BOOL ;	//Command to reset fault
  InLocal : BOOL ;	//1= Local mode (no fault by start with service switch)
  InManual : BOOL ;	//1= Manual / 0= Automatic
  InReport : BOOL ;	//Report of all state transitions
  spare0307 : BOOL ;
  InHWStop : BOOL ;	//HW stop is detected, no fault
  InDPFault : BOOL ;	//DP-Fault is detected, no fault
  InSimulation : BOOL ;	//MZAH: Simulation with DPSim
  OutComFault : BOOL ;	//Communication fault
  spare0404 : BOOL ;	//Wrong nominal values, rejected by MEAF
  spare0405 : BOOL ;	//de: Dampfventil angesteuert
  spare0406 : BOOL ;	//de: Endschalter 1 geschlossen
  spare0407 : BOOL ;	//de: Endschalter 2 geschlossen
  StOff : BOOL ;	//Element is stopped
  spare0501 : BOOL ;	//Element is starting
  StOn : BOOL ;	//Element is dosing
  spare0502 : BOOL ;	//Element is stopping
  StFault : BOOL ;	//Element has a communication or device fault
  Mill : ARRAY  [1 .. 4 ] OF STRUCT
   InEnable : BOOL ;	//1=Start Mill/0=Stop Mill
   CmdJobChange : BOOL ;	//Send new job number to MYAH
   CmdReadRegister : BOOL ;
   OutWrongValue : BOOL ;
   OutRegisterReady : BOOL ;
   OutAlarmTolMinus : BOOL ;
   OutAlarmTolPlus : BOOL ;
   OutAlarmScale : BOOL ;
   Tar : STRUCT
    RecipeNo : INT ;
    JobID : ARRAY  [1 .. 32 ] OF BYTE ;
    spare42 : INT ;
    spare44 : DINT ;
    spare48 : DINT ;
    spare52 : DINT ;
    spare56 : DINT ;
    spare60 : DINT ;
   END_STRUCT ;
   Act : STRUCT
    RecipeNo : INT ;	//[1..100]
    JobNo : DINT ;
    State : INT ;	//1=Run
    StartTime : STRUCT
     Sec : BYTE ;
     Min : BYTE ;
     Hour : BYTE ;
     Day : BYTE ;
     Month : BYTE ;
     Year : BOOL ;
    END_STRUCT ;
    TotalWeightInlet : DINT ;	//[0.1 kg or 0.1 lb]
    TotalWeightOutlet : DINT ;	//[0.1 kg or 0.1 lb]
    Flowrate : DINT ;	//[0.1 kg/g or 0.1 lb/h]
    YieldA : INT ;	//[0.00 to 200.00%]
    YieldB : INT ;	//[0.00 to 200.00%]
    AlarmNo : INT ;
    spare40 : DINT ;
    spare44 : DINT ;
    spare48 : DINT ;
    spare52 : DINT ;
    spare56 : DINT ;
    spare60 : DINT ;
   END_STRUCT ;
   Register : STRUCT
    RecipeNo : INT ;	//[1..100]
    JobNo : DINT ;
    State : INT ;	//1=Run
    StartTime : STRUCT
     Sec : BYTE ;
     Min : BYTE ;
     Hour : BYTE ;
     Day : BYTE ;
     Month : BYTE ;
     Year : BOOL ;
    END_STRUCT ;
    TotalWeightInlet : DINT ;	//[0.1 kg or 0.1 lb]
    TotalWeightOutlet : DINT ;	//[0.1 kg or 0.1 lb]
    Flowrate : DINT ;	//[0.1 kg/g or 0.1 lb/h]
    YieldA : INT ;	//[0.00 to 200.00%]
    YieldB : INT ;	//[0.00 to 200.00%]
    AlarmNo : INT ;
    spare40 : DINT ;
    spare44 : DINT ;
    spare48 : DINT ;
    spare52 : DINT ;
    spare56 : DINT ;
    spare60 : DINT ;
   END_STRUCT ;
  END_STRUCT ;
  OutAlarmNr : INT ;	//Is read from MEAF
  OutAlarmNrLog : INT ;	//Last textnumber send to log
  Par : STRUCT
   ParObjectNo : INT ;	//Is used for communication with PC, e.g. for message
   ParMsgType : INT ;	//Is used for message (translation of state)
   ParHornCode : INT ;	//Is used by horn module
   ParLogOff : BOOL ;	//Report is off
   ParManual : BOOL ;	//Manual mode wihout interlocking
   ParWithMill1 : BOOL ;
   ParWithMill2 : BOOL ;
   ParWithMill3 : BOOL ;
   ParWithMill4 : BOOL ;
   ParIOByteNr : INT ;	//PROFIBUS: Address of first input and output byte
   OutHelpFlags : STRUCT 	//Is sent to FBAL
    OutComFaultRead : BOOL ;
    OutComFaultSend : BOOL ;
    OutRelevantFault : BOOL ;
   END_STRUCT ;
   Command : STRUCT
    StartMill1 : BOOL ;	//Start/Stop Mill 1
    StartMill2 : BOOL ;	//Start/Stop Mill 2
    StartMill3 : BOOL ;	//Start/Stop Mill 3
    StartMill4 : BOOL ;	//Start/Stop Mill 4
    spare04 : BOOL ;
    spare05 : BOOL ;
    spare06 : BOOL ;
    AcceptNewDataReady : BOOL ;
    spare10 : BYTE ;
    spare20 : BYTE ;
    CommandReady : BOOL ;	//de: Steuersignale gültig
    spare31 : BOOL ;
    spare32 : BOOL ;
    spare33 : BOOL ;
    spare34 : BOOL ;
    ResetAlarm : BOOL ;	//de: Alarm löschen
    NewSendData : BOOL ;	//de: Aenderung Sendedaten
    AcceptNewRcvData : BOOL ;	//de: Quittierung Aenderung Empfangsdatensatz
   END_STRUCT ;
   Status : STRUCT
    spare00 : BOOL ;
    spare01 : BOOL ;
    spare02 : BOOL ;
    spare03 : BOOL ;
    spare04 : BOOL ;
    spare05 : BOOL ;	//
    spare06 : BOOL ;
    NewDataReady : BOOL ;	//de: Neue Werte Bereit
    spare10 : BYTE ;
    spare20 : BYTE ;
    spare30 : BOOL ;
    spare31 : BOOL ;
    spare32 : BOOL ;
    spare33 : BOOL ;	//de: Sollwertvorgabe Remote
    WrongValue : BOOL ;	//de: Falscher Sollwert
    SumFault : BOOL ;	//de: Sammelalarm
    AcceptNewSendData : BOOL ;	//de: Quittierung Aenderung Sendedaten
    NewRcvData : BOOL ;	//de: Aenderung Empfangsdaten
   END_STRUCT ;
  END_STRUCT ;
END_VAR
VAR_TEMP
  tmpLogValue : WORD ;
  tmpFault : BOOL ;
  tmpOff : BOOL ;
  tmpOn : BOOL ;
  tmpLocal : BOOL ;
  tmpLocalFault : BOOL ;
  tmpReport : BOOL ;
  tmpFlag : BOOL ;
  tmpLenDyn : DINT ;
  tmpAddr : WORD ;
  tmpReturn : INT ;
  DPData : STRUCT
   StatusCommand : DWORD ;
   NrSndDataSet : BYTE ;	//de: Nummer Sendedatensatz
   IdxSndDataSet : BYTE ;	//de: Index Sendedatensatz
   NrRcvDataSet : BYTE ;	//de: Nummer Empfangsdatensatz
   IdxRcvDataSet : BYTE ;	//de: Index Empfangsdatensatz
   Data : ARRAY  [1 .. 14 ] OF DINT ;
  END_STRUCT ;
END_VAR
BEGIN
NETWORK
TITLE =  Start Global
      L     710;
      T     #tmpLenDyn;	//--> Len dynamic data in byte
NETWORK
TITLE = PC Control
//=== Test Object number =====================
      L     "SYS_DirectCtrlDB".PC.ObjectNo;	//PCControl.ObjectNo
      L     #Par.ParObjectNo;	//Input ObjectNo
      <>I;
      JC    Ctrl;
//=== Test OType      ========================
      L     1033;	//Input object type
      L     "SYS_DirectCtrlDB".PC.ObjectType;	//PCControl.ObjectType
      <>I;
      JC    Ctrl;
//=== Test Handshake =========================
      A     "SYS_DirectCtrlDB".PC.Hsk.FExamine;	//Handshake.FExamine
      JC    pExa;
      A     "SYS_DirectCtrlDB".PC.Hsk.FDefineCmd;	//Handshake.FDefineCmd
      JC    pCmd;
      A     "SYS_DirectCtrlDB".PC.Hsk.FDefinePara;	//Handshake.FDefinePara
      JC    pPar;
pIni: L     2;	//FcInit
      UC    "SYS_DirectCtrl";
      JU    Ctrl;
//Write parameter 
pPar: NOP   0;
//Write new commands from PC to Interface of group 
pCmd: A     "SYS_DirectCtrlDB".PC.Cmd1[8];	//Cmd1[8]  =CmdOff
      S     #CmdOff;
      A     "SYS_DirectCtrlDB".PC.Cmd1[9];	//Cmd1[9]  =CmdOn
      S     #CmdOn;
      A     "SYS_DirectCtrlDB".PC.Cmd1[10];	//Cmd1[10] =CmdNext
      S     #CmdNext;
      A     "SYS_DirectCtrlDB".PC.Cmd1[11];	//Cmd1[11] =CmdFaultReset
      S     #CmdFaultReset;
      A     "SYS_DirectCtrlDB".PC.Cmd1[13];	//Cmd1[13] =CmdManualOn
      S     #InManual;
      A     "SYS_DirectCtrlDB".PC.Cmd2[13];	//Cmd2[13] =CmdManualOff
      R     #InManual;
      A     "SYS_DirectCtrlDB".PC.Cmd1[14];	//Cmd1[14] =CmdReportOn
      S     #InReport;
      A     "SYS_DirectCtrlDB".PC.Cmd2[14];	//Cmd2[14] =CmdReportOff
      R     #InReport;
//Define Value
      AN    "SYS_DirectCtrlDB".PC.Hsk.FDefineValue;	// PC.Hsk.FDefineValue
      ON    #InManual;
      JC    pIni;
      JU    pIni;
pExa: TAR2;	//Address dynamic datas
      T     "SYS_DirectCtrlDB".GC.InDynAddr;	//-->PCControl.GC.InDynAddr
      L     #tmpLenDyn;	//Length dynamic datas
      T     "SYS_DirectCtrlDB".GC.InDynLen;	//-->PCControl.GC.InDynLen
      L     0;
      T     "SYS_DirectCtrlDB".GC.InParaAddr;	//-->PCControl.GC.InParaAddr
      T     "SYS_DirectCtrlDB".GC.InParaLen;	//-->PCControl.GC.InParaLen
      L     1;	//Code FcExamine
      UC    "SYS_DirectCtrl";
      L     10;	//Revision
      T     "SYS_DirectCtrlDB".GC.Revision;
Ctrl: NOP   0;
NETWORK
TITLE = (Profibus) Read data and store Data 
      L     #Par.ParIOByteNr;
      T     #tmpAddr;
      A     #InSimulation;
      JC    rSim;
      CALL  "SIEMENS_DPRD_DAT" (
           LADDR                    := #tmpAddr,
           RET_VAL                  := #tmpReturn,
           RECORD                   := #DPData);
      L     #tmpReturn;
      L     0;
      <>I;
      =     #Par.OutHelpFlags.OutComFaultRead;
      JC    rcv0;
      JU    rDP;
//read from Simulation
rSim: R     #Par.OutHelpFlags.OutComFaultRead;
      A     "GCS7_Gr_SimDPtoImage";
      L     P#I 0.0;
      JC    rDB1;
      OPN   "TEST_IOSimuliInput";
      L     P#DBX 0.0;
rDB1: L     #Par.ParIOByteNr;
      SLD   3;
      +D;
      LAR1;
      L     D [AR1,P#0.0];
      T     #DPData.StatusCommand;
      L     B [AR1,P#4.0];
      T     #DPData.NrSndDataSet;
      L     B [AR1,P#5.0];
      T     #DPData.IdxSndDataSet;
      L     B [AR1,P#6.0];
      T     #DPData.NrRcvDataSet;
      L     B [AR1,P#7.0];
      T     #DPData.IdxRcvDataSet;
      L     D [AR1,P#8.0];
      T     #DPData.Data[1];
      L     D [AR1,P#12.0];
      T     #DPData.Data[2];
      L     D [AR1,P#16.0];
      T     #DPData.Data[3];
      L     D [AR1,P#20.0];
      T     #DPData.Data[4];
      L     D [AR1,P#24.0];
      T     #DPData.Data[5];
      L     D [AR1,P#28.0];
      T     #DPData.Data[6];
      L     D [AR1,P#32.0];
      T     #DPData.Data[7];
      L     D [AR1,P#36.0];
      T     #DPData.Data[8];
      L     D [AR1,P#40.0];
      T     #DPData.Data[9];
      L     D [AR1,P#44.0];
      T     #DPData.Data[10];
      L     D [AR1,P#48.0];
      T     #DPData.Data[11];
      L     D [AR1,P#52.0];
      T     #DPData.Data[12];
      L     D [AR1,P#56.0];
      T     #DPData.Data[13];
      L     D [AR1,P#60.0];
      T     #DPData.Data[14];
//==Copy Status===============
rDP:  L     #DPData.NrRcvDataSet;
      L     0;
      ==I;
      JC    R1_1;	//Read Dataset 1.1
      CALL  "SIEMENS_BLKMOV" (
           SRCBLK                   := #DPData.StatusCommand,
           RET_VAL                  := #tmpReturn,
           DSTBLK                   := #Par.Status);
//===============================
//Answer Dataset 1 Index1
      A(;
      L     #DPData.NrRcvDataSet;
      L     1;
      <>I;
      );
      O(;
      L     #DPData.IdxRcvDataSet;
      L     1;
      <>I;
      );
      JC    r1_2;
      CALL  "SIEMENS_BLKMOV" (
           SRCBLK                   := #DPData.Data,
           RET_VAL                  := #tmpReturn,
           DSTBLK                   := #Mill[1].Act);
      L     #tmpReturn;
      JU    R1_2;
//===============================
//Answer Dataset 1 Index 2
r1_2: A(;
      L     #DPData.NrRcvDataSet;
      L     1;
      <>I;
      );
      O(;
      L     #DPData.IdxRcvDataSet;
      L     2;
      <>I;
      );
      JC    r1_3;
      CALL  "SIEMENS_BLKMOV" (
           SRCBLK                   := #DPData.Data,
           RET_VAL                  := #tmpReturn,
           DSTBLK                   := #Mill[2].Act);
      JU    R1_3;
//===============================
//Answer Dataset 1 Index 3
r1_3: A(;
      L     #DPData.NrRcvDataSet;
      L     1;
      <>I;
      );
      O(;
      L     #DPData.IdxRcvDataSet;
      L     3;
      <>I;
      );
      JC    r1_4;
      CALL  "SIEMENS_BLKMOV" (
           SRCBLK                   := #DPData.Data,
           RET_VAL                  := #tmpReturn,
           DSTBLK                   := #Mill[3].Act);
      JU    R1_4;
//===============================
//Answer Dataset 1 Index 4
r1_4: A(;
      L     #DPData.NrRcvDataSet;
      L     1;
      <>I;
      );
      O(;
      L     #DPData.IdxRcvDataSet;
      L     4;
      <>I;
      );
      JC    r3_1;
      CALL  "SIEMENS_BLKMOV" (
           SRCBLK                   := #DPData.Data,
           RET_VAL                  := #tmpReturn,
           DSTBLK                   := #Mill[4].Act);
      JU    R3_1;
//===============================
//Answer Dataset 3 Index 1
r3_1: A(;
      L     #DPData.NrRcvDataSet;
      L     3;
      <>I;
      );
      O(;
      L     #DPData.IdxRcvDataSet;
      L     1;
      <>I;
      );
      JC    r3_2;
      S     #Mill[1].OutRegisterReady;
      R     #Mill[1].CmdReadRegister;
      CALL  "SIEMENS_BLKMOV" (
           SRCBLK                   := #DPData.Data,
           RET_VAL                  := #tmpReturn,
           DSTBLK                   := #Mill[1].Register);
      JU    R3_2;
//===============================
//Answer Dataset 3 Index 2
r3_2: A(;
      L     #DPData.NrRcvDataSet;
      L     3;
      <>I;
      );
      O(;
      L     #DPData.IdxRcvDataSet;
      L     2;
      <>I;
      );
      JC    r3_3;
      S     #Mill[2].OutRegisterReady;
      R     #Mill[2].CmdReadRegister;
      CALL  "SIEMENS_BLKMOV" (
           SRCBLK                   := #DPData.Data,
           RET_VAL                  := #tmpReturn,
           DSTBLK                   := #Mill[2].Register);
      JU    R3_2;
//===============================
//Answer Dataset 3 Index 3
r3_3: A(;
      L     #DPData.NrRcvDataSet;
      L     3;
      <>I;
      );
      O(;
      L     #DPData.IdxRcvDataSet;
      L     3;
      <>I;
      );
      JC    r3_4;
      S     #Mill[3].OutRegisterReady;
      R     #Mill[3].CmdReadRegister;
      CALL  "SIEMENS_BLKMOV" (
           SRCBLK                   := #DPData.Data,
           RET_VAL                  := #tmpReturn,
           DSTBLK                   := #Mill[3].Register);
      JU    R3_4;
//===============================
//Answer Dataset 3 Index 4
r3_4: A(;
      L     #DPData.NrRcvDataSet;
      L     3;
      <>I;
      );
      O(;
      L     #DPData.IdxRcvDataSet;
      L     4;
      <>I;
      );
      JC    R1_1;
      S     #Mill[4].OutRegisterReady;
      R     #Mill[4].CmdReadRegister;
      CALL  "SIEMENS_BLKMOV" (
           SRCBLK                   := #DPData.Data,
           RET_VAL                  := #tmpReturn,
           DSTBLK                   := #Mill[4].Register);
      JU    R1_1;
//===============================
//Read Dataset 1.1
R1_1: AN    #Par.ParWithMill1;
      JC    R1_2;
      L     1;
      T     #DPData.NrRcvDataSet;
      L     1;
      T     #DPData.IdxRcvDataSet;
      JU    rcv0;
//===============================
//Read Dataset 1.2
R1_2: AN    #Par.ParWithMill2;
      JC    R1_3;
      L     1;
      T     #DPData.NrRcvDataSet;
      L     2;
      T     #DPData.IdxRcvDataSet;
      JU    rcv0;
//===============================
//Read Dataset 1.3
R1_3: AN    #Par.ParWithMill3;
      JC    R1_4;
      L     1;
      T     #DPData.NrRcvDataSet;
      L     3;
      T     #DPData.IdxRcvDataSet;
      JU    rcv0;
//===============================
//Read Dataset 1.4
R1_4: AN    #Par.ParWithMill4;
      JC    R3_1;
      L     1;
      T     #DPData.NrRcvDataSet;
      L     4;
      T     #DPData.IdxRcvDataSet;
      JU    rcv0;
//===============================
//Read Dataset 3.1
R3_1: AN    #Par.ParWithMill1;
      ON    #Mill[1].CmdReadRegister;
      JC    R3_2;
      L     3;
      T     #DPData.NrRcvDataSet;
      L     1;
      T     #DPData.IdxRcvDataSet;
      JU    rcv0;
//===============================
//Read Dataset 3.2
R3_2: AN    #Par.ParWithMill2;
      ON    #Mill[2].CmdReadRegister;
      JC    R3_3;
      L     3;
      T     #DPData.NrRcvDataSet;
      L     2;
      T     #DPData.IdxRcvDataSet;
      JU    rcv0;
//===============================
//Read Dataset 3.3
R3_3: AN    #Par.ParWithMill3;
      ON    #Mill[3].CmdReadRegister;
      JC    R3_4;
      L     3;
      T     #DPData.NrRcvDataSet;
      L     3;
      T     #DPData.IdxRcvDataSet;
      JU    rcv0;
//===============================
//Read Dataset 3.4
R3_4: AN    #Par.ParWithMill4;
      ON    #Mill[4].CmdReadRegister;
      JC    R1_1;
      L     3;
      T     #DPData.NrRcvDataSet;
      L     4;
      T     #DPData.IdxRcvDataSet;
      JU    rcv0;
//===============================
rcv0: NOP   0;
NETWORK
TITLE = (Profibus) Status to ASW
      A     #Par.OutHelpFlags.OutComFaultRead;
      O     #Par.OutHelpFlags.OutComFaultSend;
      =     #OutComFault;
//=======================================
//Init in local mode  
//=======================================
      AN    #InLocal;
      AN    #InManual;
      ON    #OutComFault;
      JC    alJL;
alJL: NOP   0;
NETWORK
TITLE =  All State Init
//===Clear tmp Variable
//===Global Group Orders===
      A     "GCS7_Gr_OutManualOff";	//Global.OutManualOff
      R     #InManual;
      A     #InManual;
      S     "GCS7_Gr_InManual";	//Global.InManualMode
//---Report is on---
      O     "GCS7_Gr_OutReportAll";	//---Global OutReportAll
      O     #InReport;
      =     #tmpReport;
//---FaultReset is on---
      A     "GCS7_Gr_OutFaultReset";	//Gr.OutFaultReset
      S     #CmdFaultReset;
//---State---
//---Local---
      A     #InLocal;
      AN    #InManual;
      =     #tmpLocalFault;
      A     #tmpLocalFault;
      O     #InHWStop;
      O     #InDPFault;
      =     #tmpLocal;
//---Off---
      AN    #InManual;
      ON    #Par.ParManual;
      AN    #InEnable;
      O     #tmpLocal;
      O     #CmdOff;
      =     #tmpOff;
//---On---
      A     #CmdNext;
      AN    #InManual;
      O     #CmdOn;
      AN    #tmpOff;
      =     #tmpOn;
//---------
      A     #Mill[1].CmdJobChange;
      R     #Mill[1].OutRegisterReady;
//---------
      A     #Mill[2].CmdJobChange;
      R     #Mill[2].OutRegisterReady;
//---------
      A     #Mill[3].CmdJobChange;
      R     #Mill[3].OutRegisterReady;
//---------
      A     #Mill[4].CmdJobChange;
      R     #Mill[4].OutRegisterReady;
//=======================================
//Fault   
//=======================================
      L     #Mill[1].Act.AlarmNo;
      L     1;
      ==I;
      =     #Mill[1].OutAlarmTolMinus;
      L     #Mill[1].Act.AlarmNo;
      L     2;
      ==I;
      =     #Mill[1].OutAlarmTolPlus;
      L     #Mill[1].Act.AlarmNo;
      L     4;
      ==I;
      =     #Mill[1].OutAlarmScale;
//--------------------------------
      L     #Mill[2].Act.AlarmNo;
      L     1;
      ==I;
      =     #Mill[2].OutAlarmTolMinus;
      L     #Mill[2].Act.AlarmNo;
      L     2;
      ==I;
      =     #Mill[2].OutAlarmTolPlus;
      L     #Mill[2].Act.AlarmNo;
      L     4;
      ==I;
      =     #Mill[2].OutAlarmScale;
//--------------------------------
      L     #Mill[3].Act.AlarmNo;
      L     1;
      ==I;
      =     #Mill[3].OutAlarmTolMinus;
      L     #Mill[3].Act.AlarmNo;
      L     2;
      ==I;
      =     #Mill[3].OutAlarmTolPlus;
      L     #Mill[3].Act.AlarmNo;
      L     4;
      ==I;
      =     #Mill[3].OutAlarmScale;
//--------------------------------
      L     #Mill[4].Act.AlarmNo;
      L     1;
      ==I;
      =     #Mill[4].OutAlarmTolMinus;
      L     #Mill[4].Act.AlarmNo;
      L     2;
      ==I;
      =     #Mill[4].OutAlarmTolPlus;
      L     #Mill[4].Act.AlarmNo;
      L     4;
      ==I;
      =     #Mill[4].OutAlarmScale;
//--------------------------------
//--- Fault   
      A     #OutComFault;
      AN    #tmpLocal;
      =     #tmpFault;
NETWORK
TITLE = (Profibus) Prepare Command for MEAF
      NOP   0;
//==============================
      A     #Mill[1].InEnable;
      =     #Par.Command.StartMill1;
      A     #Mill[2].InEnable;
      =     #Par.Command.StartMill2;
      A     #Mill[3].InEnable;
      =     #Par.Command.StartMill3;
      A     #Mill[4].InEnable;
      =     #Par.Command.StartMill4;
//==============================
      A     #Par.Status.NewDataReady;
      =     #Par.Command.AcceptNewDataReady;
//==============================
      SET;
      =     #Par.Command.CommandReady;
//==============================
      A     #Par.Status.NewRcvData;
      =     #Par.Command.AcceptNewRcvData;
//==============================
      AN    #Par.Status.AcceptNewSendData;
      =     #Par.Command.NewSendData;
NETWORK
TITLE = (Profibus) Send Data
//======================================================
//Test Send Dataset 000 done
      L     #DPData.NrSndDataSet;
      L     0;
      <>I;
      JC    s8_1;
      JU    S8_1;	//-->send 128 Index 1
//------------------------------------------------
//Test Send Dataset 128.1 done
s8_1: L     #DPData.NrSndDataSet;
      L     128;
      <>I;
      O(;
      L     #DPData.IdxSndDataSet;
      L     1;
      <>I;
      );
      JC    s8_2;
      AN    #Par.Status.WrongValue;
      R     #Mill[1].CmdJobChange;
      S     #Mill[1].CmdReadRegister;
      A     #Par.Status.WrongValue;
      =     #Mill[1].OutWrongValue;
      JU    S8_2;	//-->Send 128 Index2
//------------------------------------------------
//Test Send Dataset 128.2 done
s8_2: L     #DPData.NrSndDataSet;
      L     128;
      <>I;
      O(;
      L     #DPData.IdxSndDataSet;
      L     2;
      <>I;
      );
      JC    s8_3;
      AN    #Par.Status.WrongValue;
      R     #Mill[2].CmdJobChange;
      S     #Mill[2].CmdReadRegister;
      A     #Par.Status.WrongValue;
      =     #Mill[2].OutWrongValue;
      JU    S8_3;	//-->Send 128 Index3
//------------------------------------------------
//Test Send Dataset 128.3 done
s8_3: L     #DPData.NrSndDataSet;
      L     128;
      <>I;
      O(;
      L     #DPData.IdxSndDataSet;
      L     3;
      <>I;
      );
      JC    s8_4;
      AN    #Par.Status.WrongValue;
      R     #Mill[3].CmdJobChange;
      S     #Mill[3].CmdReadRegister;
      A     #Par.Status.WrongValue;
      =     #Mill[3].OutWrongValue;
      JU    S8_4;	//-->Send 128 Index4
//------------------------------------------------
//Test Send Dataset 128.4 done
s8_4: L     #DPData.NrSndDataSet;
      L     128;
      <>I;
      O(;
      L     #DPData.IdxSndDataSet;
      L     4;
      <>I;
      );
      JC    S8_1;
      AN    #Par.Status.WrongValue;
      R     #Mill[4].CmdJobChange;
      S     #Mill[4].CmdReadRegister;
      A     #Par.Status.WrongValue;
      =     #Mill[4].OutWrongValue;
      JU    S8_1;	//-->Send 128 Index1
//==================================================
//Send Dataset 128.1
S8_1: AN    #Mill[1].CmdJobChange;
      JC    S8_2;
      L     128;
      T     #DPData.NrSndDataSet;
      L     1;
      T     #DPData.IdxSndDataSet;
      CALL  "SIEMENS_BLKMOV" (
           SRCBLK                   := #Mill[1].Tar,
           RET_VAL                  := #tmpReturn,
           DSTBLK                   := #DPData.Data);
      JU    Snd;
//==================================================
//Send Dataset 128.2
S8_2: AN    #Mill[2].CmdJobChange;
      JC    S8_3;
      L     128;
      T     #DPData.NrSndDataSet;
      L     2;
      T     #DPData.IdxSndDataSet;
      CALL  "SIEMENS_BLKMOV" (
           SRCBLK                   := #Mill[2].Tar,
           RET_VAL                  := #tmpReturn,
           DSTBLK                   := #DPData.Data);
      JU    Snd;
//==================================================
//Send Dataset 128.3
S8_3: AN    #Mill[3].CmdJobChange;
      JC    S8_4;
      L     128;
      T     #DPData.NrSndDataSet;
      L     3;
      T     #DPData.IdxSndDataSet;
      CALL  "SIEMENS_BLKMOV" (
           SRCBLK                   := #Mill[3].Tar,
           RET_VAL                  := #tmpReturn,
           DSTBLK                   := #DPData.Data);
      JU    Snd;
//==================================================
//Send Dataset 128.4
S8_4: AN    #Mill[4].CmdJobChange;
      JC    S000;
      L     128;
      T     #DPData.NrSndDataSet;
      L     4;
      T     #DPData.IdxSndDataSet;
      CALL  "SIEMENS_BLKMOV" (
           SRCBLK                   := #Mill[4].Tar,
           RET_VAL                  := #tmpReturn,
           DSTBLK                   := #DPData.Data);
      JU    Snd;
//======================================================
//Send Dataset 0
S000: L     0;
      T     #DPData.NrSndDataSet;
      L     0;
      T     #DPData.IdxSndDataSet;
//======================================================
//Senden DP
Snd:  CALL  "SIEMENS_BLKMOV" (
           SRCBLK                   := #Par.Command,
           RET_VAL                  := #tmpReturn,
           DSTBLK                   := #DPData.StatusCommand);
      A     #InSimulation;
      JC    sSim;
      CALL  "SIEMENS_DPWR_DAT" (
           LADDR                    := #tmpAddr,
           RECORD                   := #DPData,
           RET_VAL                  := #tmpReturn);
      L     #tmpReturn;
      L     0;
      <>I;
      =     #Par.OutHelpFlags.OutComFaultSend;
      JU    sEnd;
//write to Simulation
sSim: R     #Par.OutHelpFlags.OutComFaultSend;
      A     "GCS7_Gr_SimDPtoImage";
      L     P#Q 0.0;
      JC    rDB2;
      OPN   "TEST_IOSimuliOutput";
      L     P#DBX 0.0;
rDB2: L     #Par.ParIOByteNr;
      SLD   3;
      +D;
      LAR1;
      L     #DPData.StatusCommand;
      T     D [AR1,P#0.0];
      L     #DPData.NrSndDataSet;
      T     B [AR1,P#4.0];
      L     #DPData.IdxSndDataSet;
      T     B [AR1,P#5.0];
      L     #DPData.NrRcvDataSet;
      T     B [AR1,P#6.0];
      L     #DPData.IdxRcvDataSet;
      T     B [AR1,P#7.0];
      L     #DPData.Data[1];
      T     D [AR1,P#8.0];
      L     #DPData.Data[2];
      T     D [AR1,P#12.0];
      L     #DPData.Data[3];
      T     D [AR1,P#16.0];
      L     #DPData.Data[4];
      T     D [AR1,P#20.0];
      L     #DPData.Data[5];
      T     D [AR1,P#24.0];
      L     #DPData.Data[6];
      T     D [AR1,P#28.0];
      L     #DPData.Data[7];
      T     D [AR1,P#32.0];
      L     #DPData.Data[8];
      T     D [AR1,P#36.0];
      L     #DPData.Data[9];
      T     D [AR1,P#40.0];
      L     #DPData.Data[10];
      T     D [AR1,P#44.0];
      L     #DPData.Data[11];
      T     D [AR1,P#48.0];
      L     #DPData.Data[12];
      T     D [AR1,P#52.0];
      L     #DPData.Data[13];
      T     D [AR1,P#56.0];
      L     #DPData.Data[14];
      T     D [AR1,P#60.0];
sEnd: NOP   0;
NETWORK
TITLE = States
//===State machine===
      A     #StOff;
      JC    S0;
      A     #StOn;
      JC    S2;
      A     #StFault;
      JC    S4;
      S     #StOff;	//Init
      JU    S0;
NETWORK
TITLE =  StOff
xxS0: S     #StOff;
      R     #StOn;
      JU    LOGX;
S0:   A     #tmpFault;
      R     #StOff;
      JC    xxS4;	//--> Transition to StFault
      AN    #OutComFault;
      A     #tmpOn;
      R     #StOff;
      JC    xxS2;	//--> Transition to StOn
      JU    OUT;
NETWORK
TITLE =  StStarted
xxS2: S     #StOn;
      JU    LOGX;
S2:   A     #tmpFault;	//Condition for StFault/StFalse
      R     #StOn;
      JC    xxS4;	//--> Transition to StFault
      A     #tmpOff;
      R     #StOff;
      JC    xxS0;	//--> Transition to StStOff
      JU    OUT;
NETWORK
TITLE =  FAULT
// State Fault
S4:   AN    #tmpFault;	//---Condition for StOff
      A     #CmdFaultReset;
      O     #tmpLocalFault;
      R     #StFault;
      S     #StOff;
      JC    LOGC;	// Transition to StOff
      A     #tmpFault;
      A     #CmdFaultReset;
      JC    xxS4;
      JU    OUT;
NETWORK
TITLE = LOG
      L     B#(4, 0);	// Message ('Off')
      A     #StOff;
      A     #InReport;
      JC    LOG;
      L     B#(4, 1);	// Message ('On')
      A     #StOn;
      A     #InReport;
      JC    LOG;
      JU    OUT;
xxS4: S     "GCS7_Gr_InFaultFlag";	//Gr.InFaultFlag
      S     #StFault;
      CALL  "SYS_Horn_Code" (
           FcCode                   := 1,
           ParObjectType            := 1033,
           ParObjectNo              := #Par.ParObjectNo,
           ParHornCode              := #Par.ParHornCode);
//Alarm Communication
      L     B#(4, 15);	// Message ('fault communication' )
      A     #OutComFault;
      JU    LOG;
//===============================================
//State Transition
LOGX: AN    #tmpReport;
      JC    OUT;
      A     #StOff;
      L     B#(4, 1);	//Message ('Off')
      JC    LOG;
      A     #StOn;
      L     B#(4, 2);	//Message ('On')
      JC    LOG;
      JU    OUT;
LOGC: L     B#(3, 9);	//Message Operator ('fault cancelled' )
LOG:  A     #Par.ParLogOff;	//---Set LOG Message
      JC    OUT;
      T     #tmpLogValue;
      L     W#16#FF;
      AW;
      T     #OutAlarmNrLog;
      CALL  "GCS7_LogConvert" (
           ObjectNo                 := #Par.ParObjectNo,
           MsgType                  := #Par.ParMsgType,
           ClassMsgTxt              := #tmpLogValue,
           OType                    := 1033);	//LOG Message Converter / Entry / Contains Class and TextNo
NETWORK
TITLE = Global End
OUT:  SET;	//---Clear all commands
      R     #CmdOff;
      R     #CmdOn;
      R     #CmdNext;
      R     #CmdFaultReset;
//--Output for group 
      AN    #InLocal;
      O     #InManual;
      A     #InDPFault;
      S     "GCS7_Gr_InDPFault";
      AN    #InLocal;
      O     #InManual;
      A     #InHWStop;
      S     "GCS7_Gr_InHWStop";
NETWORK
TITLE = State Code
//--Stopped, Substate ---
      AN    #StOff;
      JC    STC2;
      L     41;	//Code: StOff.HWStop
      A     #InHWStop;
      JC    STC;
      L     51;	//Code: StOff.DPFault
      A     #InDPFault;
      JC    STC;
      L     1;	//Code: StOff
      JC    STC;
//--------------------
STC2: L     3;	//Code: StOn
      A     #StOn;
      JC    STC;
      L     32;	//Code: fault
STC:  L     #StCode;	//Old state code
      TAK;
      T     #StCode;	//Save state code
      <>I;
      L     3;	//Load code for CBit methode
      CC    "SYS_CBitCtrl";
END_FUNCTION_BLOCK

